Staubli VAL3: partNum.pgx

program partNum()
  local num i
  local num l_n
  local num l_ndis
begin
  //  l_n=(size(pCircle)-1)/2
  //  while l_n<size(nPartdis)
  //    $ddel(nPartdis,size(nPartdis)-1)
  //    $ddel(nPartNum,size(nPartNum)-1)
  //  endWhile
  //  while l_n>size(nPartdis)
  //    $dins(nPartdis,size(nPartdis))
  //    $dins(nPartNum,size(nPartNum))
  //  endWhile
  //  for i=0 to l_n-1
  //    nPartdis[i]=distance(pCircle[2*i].trsf,pCircle[2*i+1].trsf)+distance(pCircle[2*i+2].trsf,pCircle[2*i+1].trsf)
  //    l_ndis=l_ndis+nPartdis[i]
  //  endFor
  //  for i=0 to l_n-1
  //    nPartNum[i]=round(nPointnum*nPartdis[i]/l_ndis)
  //  endFor
end
